// TIA Portal project "Ex3-PusherGame" (V15.1)

(* hardware
DEVICE "S7-1200 station_1"  S7-1200 Station
   slot 0: "Rack_0"  S7-1200 Rack  Rack  V1.0
   slot 1: "PLC_1"  CPU 1214C AC/DC/Rly  6ES7 214-1BG31-0XB0  V3.0
*)

// ===== PLC "PLC_1"  CPU 1214C AC/DC/Rly =====

VAR_GLOBAL   // PLC tag table "Default tag table"
   "Clock_Byte" AT %MB255 : Byte;
   "Clock_10Hz" AT %M255.0 : Bool;
   "Clock_5Hz" AT %M255.1 : Bool;
   "Clock_2.5Hz" AT %M255.2 : Bool;
   "Clock_2Hz" AT %M255.3 : Bool;
   "Clock_1.25Hz" AT %M255.4 : Bool;
   "Clock_1Hz" AT %M255.5 : Bool;
   "Clock_0.625Hz" AT %M255.6 : Bool;
   "Clock_0.5Hz" AT %M255.7 : Bool;
   "System_Byte" AT %MB254 : Byte;
   "FirstScan" AT %M254.0 : Bool;
   "DiagStatusUpdate" AT %M254.1 : Bool;
   "AlwaysTRUE" AT %M254.2 : Bool;
   "AlwaysFALSE" AT %M254.3 : Bool;
   "mPoClock_10Hz" AT %M254.5 : Bool;
END_VAR

VAR_GLOBAL   // PLC tag table "Tag table_FIO"
   "iPSH1_SenOut_S11" AT %I0.0 : Bool;   // Pusher 1 - Sensor pusher out
   "iPSH1_SenIn_S12" AT %I0.1 : Bool;   // Pusher 1 - Sensor pusher in
   "iPSH2_SenOut_S21" AT %I0.2 : Bool;   // Pusher 2 - Sensor pusher out
   "iPSH2_SenIn_S22" AT %I0.3 : Bool;   // Pusher 2 - Sensor pusher in
   "iPSH3_SenOut_S31" AT %I0.4 : Bool;   // Pusher 3 - Sensor pusher out
   "iPSH3_SenIn_S32" AT %I0.5 : Bool;   // Pusher 3 - Sensor pusher in
   "iPSH4_SenOut_S41" AT %I0.6 : Bool;   // Pusher 4 - Sensor pusher out
   "iPSH4_SenIn_S42" AT %I0.7 : Bool;   // Pusher 4 - Sensor pusher in
   "iCC_BtnStart_S1" AT %I1.0 : Bool;   // Button on control cabinet - Start
   "iCC_BtnStop_S2" AT %I1.1 : Bool;   // Button on control cabinet - Stop
   "iCC_BtnReset_S3" AT %I1.2 : Bool;   // Button on control cabinet - Reset
   "iFIO_BtnReset" AT %I1.7 : Bool;   // Reset scene from Factory IO
   "oPSH1_VlvOut_K11" AT %Q0.0 : Bool;   // Pusher 1 - Move pusher out
   "oPSH2_VlvOut_K21" AT %Q0.1 : Bool;   // Pusher 2 - Move pusher out
   "oPSH3_VlvOut_K31" AT %Q0.2 : Bool;   // Pusher 3 - Move pusher out
   "oPSH3_VlvIn_K32" AT %Q0.3 : Bool;   // Pusher 3 - Move pusher in
   "oCC_LmpStart_H1" AT %Q1.0 : Bool;   // Lamp on control cabinet - Start
   "oCC_LampErr_H2" AT %Q1.1 : Bool;   // Lamp on control cabinet - Error
   "iPSH4_PV" AT %ID100 : Real;   // Pusher 4 - Process value
   "iCC_PotSpd_R1" AT %ID104 : Real;   // Pot. meter on control cabinet - Speed control
   "oPSH4_SP" AT %QD100 : Real;   // Pusher 4 - Setpoint
   "oCC_DisRounds" AT %QD104 : DInt;   // Display on control cabinet - Number of rounds
END_VAR

VAR_GLOBAL   // PLC tag table "Tag table_Flags"
   "mCam" AT %MD0 : Real;   // Virtual cam
   "mStarted" AT %M8.0 : Bool;   // Game started
   "mPoStarted" AT %M8.1 : Bool;   // Positive edge on game started
   "mRounds" AT %MW4 : Int;   // Number of rounds
   "mCC_PotSpd" AT %MD6 : Real;   // Pot. meter speed as REAL
   "mAL_PSH1Out" AT %M10.0 : Bool;   // Alarm - Pusher 1 sensor out (+)
   "mAL_PSH1In" AT %M10.1 : Bool;   // Alarm - Pusher 1 sensor in (-)
   "mAL_PSH2Out" AT %M10.2 : Bool;   // Alarm - Pusher 2 sensor out (+)
   "mAL_PSH2In" AT %M10.3 : Bool;   // Alarm - Pusher 2 sensor in (-)
   "mAL_PSH3Out" AT %M10.4 : Bool;   // Alarm - Pusher 3 sensor out (+)
   "mAL_PSH3In" AT %M10.5 : Bool;   // Alarm - Pusher 3 sensor in (-)
   "mAL_PSH4Out" AT %M10.6 : Bool;   // Alarm - Pusher 4 sensor out (+)
   "mAL_PSH4In" AT %M10.7 : Bool;   // Alarm - Pusher 4 sensor in (-)
END_VAR

// folder: System blocks/Program resources

DATA_BLOCK "ID_TON_Started"   // DB1
{ S7_Optimized_Access := 'TRUE' }
AUTHOR : Simatic
FAMILY : IEC
NAME : IEC_TMR
VERSION : 1.0
// stored: InstanceOfName IEC_TIMER
"IEC_TIMER"
BEGIN
END_DATA_BLOCK

// folder: (top level)

FUNCTION "FC_CC" : Void   // FC1, FBD
TITLE = Control cabinet
{ S7_Optimized_Access := 'TRUE' }
VERSION : 0.1
BEGIN

REGION Network 1: Start-stop
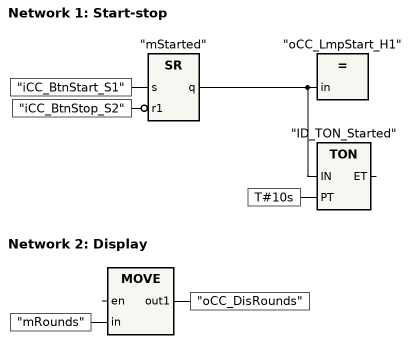
   IF "iCC_BtnStart_S1" THEN
       "mStarted" := TRUE;   // SR flip-flop
   END_IF;
   IF NOT "iCC_BtnStop_S2" THEN "mStarted" := FALSE; END_IF;
   "oCC_LmpStart_H1" := "mStarted";
   "ID_TON_Started".TON(IN := "mStarted", PT := T#10s);
END_REGION

REGION Network 2: Display
   "oCC_DisRounds" := "mRounds";
END_REGION
END_FUNCTION

FUNCTION "FC_CamController" : Void   // FC2, FBD
TITLE = Cam Controller
{ S7_Optimized_Access := 'TRUE' }
VERSION : 0.1
   VAR_TEMP   // added for the SCL form of the ladder/FBD networks
      _w1 : Bool;
   END_VAR
BEGIN

REGION Network 1: Reset Cam when started
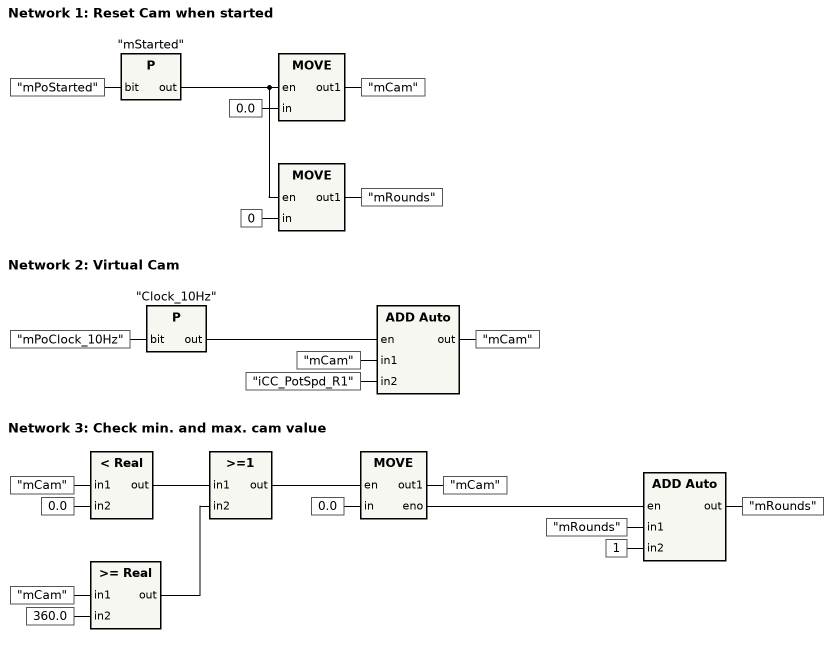
   #_w1 := "mStarted" AND NOT "mPoStarted";   // rising edge of "mStarted"
   "mPoStarted" := "mStarted";
   IF #_w1 THEN
       "mCam" := 0.0;
       "mRounds" := 0;
   END_IF;
END_REGION

REGION Network 2: Virtual Cam
   // Cam turns around from 0°to 359°
   #_w1 := "Clock_10Hz" AND NOT "mPoClock_10Hz";   // rising edge of "Clock_10Hz"
   "mPoClock_10Hz" := "Clock_10Hz";
   IF #_w1 THEN "mCam" := "mCam" + "iCC_PotSpd_R1"; END_IF;
END_REGION

REGION Network 3: Check min. and max. cam value
   // Min. value = 0°
   // Max. value = 359,99°
   // ENO of a box is taken as its EN; it also drops when the box reports an error
   #_w1 := ("mCam" < 0.0) OR ("mCam" >= 360.0);
   IF #_w1 THEN
       "mCam" := 0.0;
       "mRounds" := "mRounds" + 1;
   END_IF;
END_REGION
END_FUNCTION

FUNCTION "FC_Pusher1" : Void   // FC3, FBD
TITLE = Pusher 1
{ S7_Optimized_Access := 'TRUE' }
VERSION : 0.1
BEGIN

REGION Network 1: Pusher out
   // IF 0° > Cam > 45°
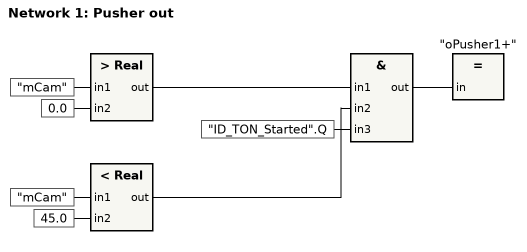
   "oPusher1+" := ("mCam" > 0.0) AND ("mCam" < 45.0) AND "ID_TON_Started".Q;
END_REGION

REGION Network 2: Pusher in
   // IF 45° > Cam > 90°
END_REGION
END_FUNCTION

FUNCTION "FC_Pusher2" : Void   // FC4, FBD
TITLE = Pusher 2
{ S7_Optimized_Access := 'TRUE' }
VERSION : 0.1
BEGIN

REGION Network 1: Pusher out
   // IF 90° > Cam > 135°
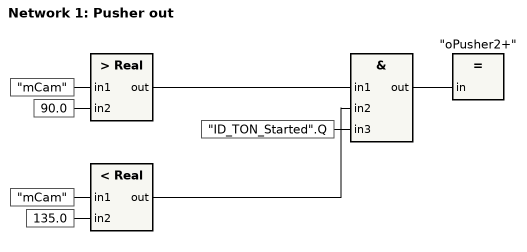
   "oPusher2+" := ("mCam" > 90.0) AND ("mCam" < 135.0) AND "ID_TON_Started".Q;
END_REGION

REGION Network 2: Pusher in
   // IF 135° > Cam > 180°
END_REGION
END_FUNCTION

FUNCTION "FC_Pusher3" : Void   // FC5, FBD
TITLE = Pusher 3
{ S7_Optimized_Access := 'TRUE' }
VERSION : 0.1
BEGIN

REGION Network 1: Pusher out
   // IF 180° > Cam > 225°
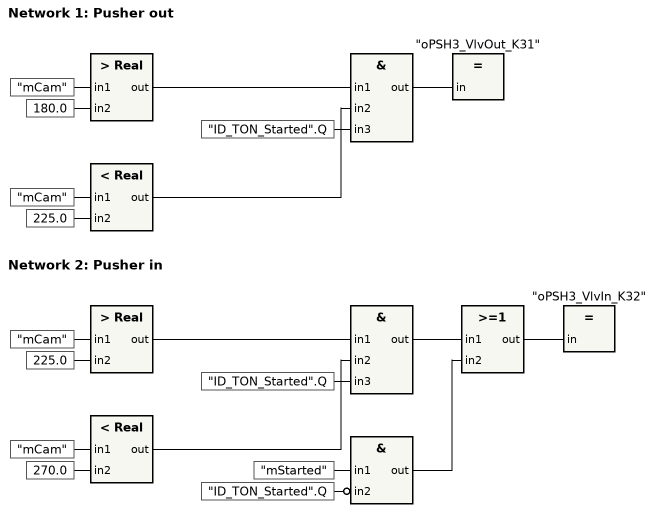
   "oPSH3_VlvOut_K31" := ("mCam" > 180.0) AND ("mCam" < 225.0) AND "ID_TON_Started".Q;
END_REGION

REGION Network 2: Pusher in
   // IF 225° > Cam > 270°
   "oPSH3_VlvIn_K32" := (("mCam" > 225.0) AND ("mCam" < 270.0) AND "ID_TON_Started".Q) OR ("mStarted" AND NOT "ID_TON_Started".Q);
END_REGION
END_FUNCTION

FUNCTION "FC_Pusher4" : Void   // FC6, FBD
TITLE = Pusher 4
{ S7_Optimized_Access := 'TRUE' }
VERSION : 0.1
BEGIN

REGION Network 1: Not started
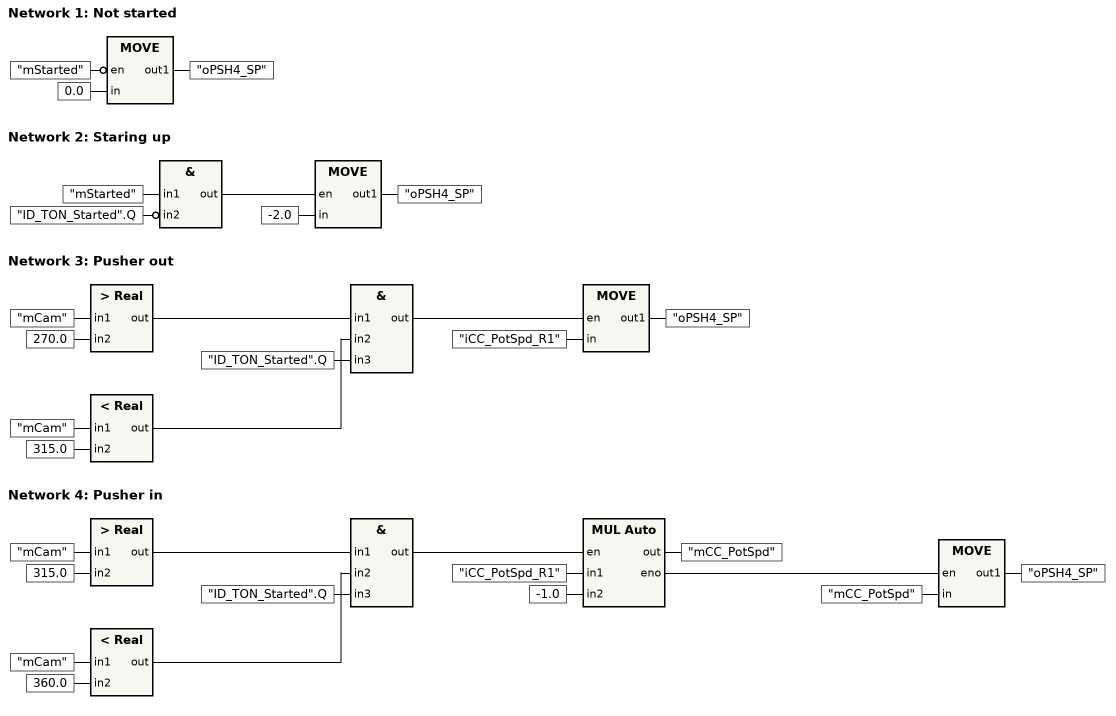
   IF NOT "mStarted" THEN "oPSH4_SP" := 0.0; END_IF;
END_REGION

REGION Network 2: Staring up
   // Go to start position
   IF "mStarted" AND NOT "ID_TON_Started".Q THEN "oPSH4_SP" := -2.0; END_IF;
END_REGION

REGION Network 3: Pusher out
   // IF 270° > Cam > 315°
   IF ("mCam" > 270.0) AND ("mCam" < 315.0) AND "ID_TON_Started".Q THEN
       "oPSH4_SP" := "iCC_PotSpd_R1";
   END_IF;
END_REGION

REGION Network 4: Pusher in
   // IF 315° > Cam > 360°
   // ENO of a box is taken as its EN; it also drops when the box reports an error
   IF ("mCam" > 315.0) AND ("mCam" < 360.0) AND "ID_TON_Started".Q THEN
       "mCC_PotSpd" := "iCC_PotSpd_R1" * (-1.0);
       "oPSH4_SP" := "mCC_PotSpd";
   END_IF;
END_REGION
END_FUNCTION

ORGANIZATION_BLOCK "Main"   // OB1, FBD, ProgramCycle
TITLE = "Main Program Sweep (Cycle)"
{ S7_Optimized_Access := 'TRUE' }
VERSION : 0.1
BEGIN

REGION Network 1: Control cabinet
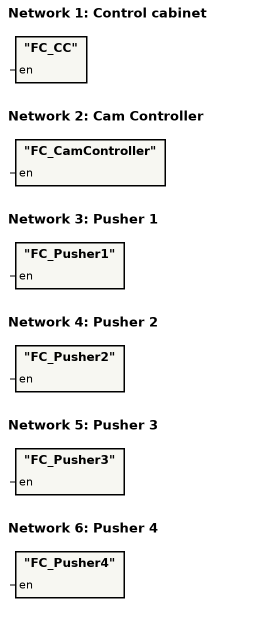
   "FC_CC"();
END_REGION

REGION Network 2: Cam Controller
   "FC_CamController"();
END_REGION

REGION Network 3: Pusher 1
   "FC_Pusher1"();
END_REGION

REGION Network 4: Pusher 2
   "FC_Pusher2"();
END_REGION

REGION Network 5: Pusher 3
   "FC_Pusher3"();
END_REGION

REGION Network 6: Pusher 4
   "FC_Pusher4"();
END_REGION
END_ORGANIZATION_BLOCK